FUNCTION_BLOCK PixelVideoClass EXTENDS FB_CyclicFB IMPLEMENTS ITF_Video
VAR
	CurrentFrame: INT := 0;
	TotalFramesInFilm: INT;
	ThisVideo: ARRAY[0..99, 0..255] OF UDINT;
	I: INT;
END_VAR

METHOD GetNextFrame : ARRAY[0..255] OF UDINT
FOR I := 0 TO 255 DO
	GetNextFrame[I] := ThisVideo[CurrentFrame,I];
END_FOR

IF CurrentFrame = TotalFramesInFilm - 1 THEN
	CurrentFrame := 0;
ELSE
	CurrentFrame := CurrentFrame + 1;
END_IF
END_METHOD

END_FUNCTION_BLOCK

(* stored: Version 1.1.0.1, ProductVersion 3.1.4024.13
   POU PixelVideoClass: Id {cc90f7c9-29e6-479a-b84c-aa032a257c67}, SpecialFunc None
   Method GetNextFrame: Id {26e244c8-5196-4630-95f7-ff67685fbedb} *)
